TYPE ST_Sample :
STRUCT
	nCounter : INT;
	bReady : BOOL;
	aIntArray : ARRAY[0..50] OF INT;  
END_STRUCT
END_TYPE

(* stored: Version 1.1.0.1, ProductVersion 3.1.4024.13
   DUT ST_Sample: Id {0c2ae62b-4655-4256-ab69-92b52ee3edda} *)
